   		If rst.Fields(8).Value <> 0 And rst.Fields(7).Value <> 0 Then ' Si el ciclo es no valido
   
   
   		VarC	= CInt(rst.Fields(6).Value) / 10
   		VarPR	= CInt(rst.Fields(7).Value)
   		
   		bfde4b54-0db7-4817-8032-87127bf19bb9 "VarC# " & VarC & " y VarPR " & VarPR
   			
   		
   			' Suma de formulas utilizadas
   			If LavadoraNro <> 4 Then
   				programaBraun(VarPR) = programaBraun(VarPR) + 1
   		If Err.Number <> 0 Then
   			bfde4b54-0db7-4817-8032-87127bf19bb9 "Error en S500 - en la asignacion de variables programaBraun en loop#" & Err.Number & " " & Err.Description
   			Err.Clear
   			Set conn = Nothing  
   			Exit Sub
   		End If
   				tCargaBraun(VarPR) = tCargaBraun(VarPR) + VarC
   		If Err.Number <> 0 Then
   			bfde4b54-0db7-4817-8032-87127bf19bb9 "Error en S500 - en la asignacion de variables tCargaBraun en loop#" & Err.Number & " " & Err.Description
   			Err.Clear
   			Set conn = Nothing  
   			Exit Sub
   		End If
   			Else
   				programaGirbau(VarPR) = programaGirbau(VarPR) + 1
   		If Err.Number <> 0 Then
   			bfde4b54-0db7-4817-8032-87127bf19bb9 "Error en S500 - en la asignacion de variables programaGirbau en loop#" & Err.Number & " " & Err.Description
   			Err.Clear
   			Set conn = Nothing  
   			Exit Sub
   		End If
   				tCargaGirbau(VarPR) = tCargaGirbau(VarPR) + VarC
   		If Err.Number <> 0 Then
   			bfde4b54-0db7-4817-8032-87127bf19bb9 "Error en S500 - en la asignacion de variables tCargaGirbau en loop#" & Err.Number & " " & Err.Description
   			Err.Clear
   			Set conn = Nothing  
   			Exit Sub
   		End If
   			End If
   			
   		End If
   		
   		rst.MoveNext
   		
   		If Err.Number <> 0 Then
   			bfde4b54-0db7-4817-8032-87127bf19bb9 "Error en S500 - en la asignacion de variables locales en loop#" & Err.Number & " " & Err.Description
   			Err.Clear
   			Set conn = Nothing  
   			Exit Sub
   		End If
   	Loop
   	
   	bfde4b54-0db7-4817-8032-87127bf19bb9 "Sale del loop de Lectura de registros S500 - de Lav nro " & LavadoraNro
   	
   	conn.close
   	Set rst = Nothing
   	Set conn = Nothing
   	
   Next
   
   bfde4b54-0db7-4817-8032-87127bf19bb9 "Sale del loop general de rst"
   
   '' %%%%%%%%%%%%%%%%%%%%%%%%%%%%%%%%%%%%%%%%%%%%%%%%%%%%%%%%%%%%%%%%%%%%%%%%%%%%%%%%%%%%%%%%%%%%%%%%%%%%%%%%%%%
   '' %%%%%%%%%%%%    IMPRESION DE DATOS EN INFORME    %%%%%%%%%%%%%%%%%%%%%%%%  XD  %%%%%%%%%%%%%%%%%%%%%%%%%%%%
   '' %%%%%%%%%%%%%%%%%%%%%%%%%%%%%%%%%%%%%%%%%%%%%%%%%%%%%%%%%%%%%%%%%%%%%%%%%%%%%%%%%%%%%%%%%%%%%%%%%%%%%%%%%%%
   
   Dim NameInfDiario
   
   
   If Err.Number <> 0 Then
   	bfde4b54-0db7-4817-8032-87127bf19bb9 "Cambio de nombre Informe Diario Lavs S500 - 2 Error #" & Err.Number & " " & Err.Description
   	Err.Clear 
   	Exit Sub
   End If
   
   ' Creacion devariables locales
   Dim objExcel
   Dim colMaquinadosBraun, colCantidadesBraun, colMaquinadosGirbau, colCantidadesGirbau
   Dim objfso
   
   'Asignacion inicial de variables locales
   colMaquinadosBraun	= 3
   colMaquinadosGirbau = 9
   colCantidadesBraun	= 4
   colCantidadesGirbau	= 10
   	
   'Creacion de Archivo .xls
   Set objExcel = CreateObject("Excel.Application")
   
   objExcel.Visible = False
   
   objExcel.Workbooks.Open "C:\ESPACIO DE TRABAJO\InformeDiario\Plantillas\InformeDiarioLavsMensual.xls"
   
   'Fin creacion archivo .xls
   If Err.Number <> 0 Then
   	bfde4b54-0db7-4817-8032-87127bf19bb9 "Error en  creacion de archivo: " & Err.Number & " :" & Err.Description
   	Err.Clear
   End If
   
   ' Imprimo tipo de informe
   objExcel.Cells(2,5).Value = impTipo
   
   objExcel.Cells(3,5).Value = impDesde
   objExcel.Cells(3,8).Value = impHasta
   						
   ' Inserción de datos en el informe
   
   'Datos de cantidad de programas
   For i = 0 To 14
   	
   	If i <= 9 Then
   		objExcel.Cells(i+7,colMaquinadosBraun).Value 	= programaBraun		(i + 1)
   		objExcel.Cells(i+7,colCantidadesBraun).Value 	= tCargaBraun		(i + 1)
   		objExcel.Cells(i+7,colMaquinadosGirbau).Value 	= programaGirbau	(i + 1)
   		objExcel.Cells(i+7,colCantidadesGirbau).Value 	= tCargaGirbau		(i + 1)
   	End If
   	
   If Err.Number <> 0 Then
   	bfde4b54-0db7-4817-8032-87127bf19bb9 "Error en Impresion de formulas 1ra en: " & i & " #" & Err.Number & " " & Err.Description
   	Err.Clear
   End If
   	
   	If i > 9 And i <= 11 Then
   		objExcel.Cells(i+12,colMaquinadosBraun).Value	= programaBraun		(i + 1)
   		objExcel.Cells(i+12,colCantidadesBraun).Value	= tCargaBraun		(i + 1)
   		objExcel.Cells(i+12,colMaquinadosGirbau).Value	= programaGirbau	(i + 1)
   		objExcel.Cells(i+12,colCantidadesGirbau).Value	= tCargaGirbau		(i + 1)
   	End If
   	
   If Err.Number <> 0 Then
   	bfde4b54-0db7-4817-8032-87127bf19bb9 "Error en Impresion de formulas 2da en: " & i & " #" & Err.Number & " " & Err.Description
   	Err.Clear
   End If
   	
   	If i > 11 Then
   		objExcel.Cells(i+5,colMaquinadosBraun).Value 	= programaBraun		(i + 1)
   		objExcel.Cells(i+5,colCantidadesBraun).Value 	= tCargaBraun		(i + 1)
   		objExcel.Cells(i+5,colMaquinadosGirbau).Value 	= programaGirbau	(i + 1)
   		objExcel.Cells(i+5,colCantidadesGirbau).Value 	= tCargaGirbau		(i + 1)
   		
   	End If
   	
   If Err.Number <> 0 Then
   	bfde4b54-0db7-4817-8032-87127bf19bb9 "Error en Impresion de formulas 3ra en: " & i & " #" & Err.Number & " " & Err.Description
   	Err.Clear
   End If
   Next
   
   If Err.Number <> 0 Then
   	bfde4b54-0db7-4817-8032-87127bf19bb9 "Error en Impresion de formulas#" & Err.Number & " " & Err.Description
   	Err.Clear
   End If
   
   ' Fin de impresion de datos en tabla
   Dim Text
   Select Case tipo_Inf
   	Case 0 ' Periodico
   		Text = "Informe_Periodico"
   	Case 1
   		Text = "Informe_Mensual"
   	Case 2
   		Text = "Informe_Anual"	
   End Select
   
   NameInfDiario = "C:\ESPACIO DE TRABAJO\InformeDiario\" & Text & "_Lavs" &(Replace(CStr(Date),"/","")&Replace(CStr(Time),":",""))&".xls"
   
   objExcel.ActiveWorkbook.SaveAs NameInfDiario, 56
   objExcel.ActiveWorkbook.Close
   objExcel.Application.Quit
   
   
   Set objfso = CreateObject("Scripting.FileSystemObject")
   Do While objfso.FileExists(NameInfDiario) = False
   Loop
   k = Timer +5
   Do While (Timer<k)
   Loop	
   
   	If Err.Number <> 0 Then
   		bfde4b54-0db7-4817-8032-87127bf19bb9 "Error en creacion de archivo excel#" & Err.Number & " " & Err.Description
   		Err.Clear
   	End If
   
   bfde4b54-0db7-4817-8032-87127bf19bb9 "NameInfDiario#" & CStr(NameInfDiario)
   
   '## ENVIAR INFORME POR EMAIL
   
   Dim appOutlook 'As OUTLOOK.APPLICATION
   Dim mlNewMail 'As MailItem
   Dim objEntry
   
   
   Const addressee = "crj@eprocsrl.com.ar; danielst@live.com.ar; josemariacullen@hotmail.com;"' zekeserio@hotmail.com;"
   
   Set appOutlook = CreateObject("OUTLOOK.APPLICATION")
   
   
   'Generating and sending an e-mail:
   Set mlNewMail = appOutlook.CreateItem(0)
   mlNewMail.Display
   mlNewMail.To = addressee
   mlNewMail.Subject = Text + " de produccion"
   mlNewMail.Body = Text
   
   mlNewMail.Attachments.Add CStr(NameInfDiario)
   
   mlNewMail.save
   mlNewMail.send 
   
   'Error routine
   If Err.Number <> 0 Then
   	bfde4b54-0db7-4817-8032-87127bf19bb9 "Error al enviar el email #" & Err.Number & " " & Err.Description
   End If

VB script "S404_ActMes"
   	Dim mesAnterior
   
   	mesAnterior = Date()
   
   	mesAnterior = DateAdd("m",-1, mesAnterior)
   	
   	SmartTags("Inf_Mes") = Month(mesAnterior)
   	

VB script "S405_ActAno"
   	Dim anoAnterior
   
   	anoAnterior = Date()
   
   	anoAnterior = DateAdd("yyyy",-1, anoAnterior)
   	
   	SmartTags("Inf_Ano") = Year(anoAnterior)
   	

VB script "S406_UltimoDiaDelMes"
   Dim bisiesto
   
   ' verificar que el año sea bisiesto
   If (ano Mod 4) = 0 And ((ano Mod 100) <> 0 Or (ano Mod 400) = 0) Then
   	bisiesto = 1
   Else
   	bisiesto = 0
   End If
   
   If mes = 1 Or mes = 3 Or mes = 5 Or mes = 7 Or mes = 8 Or mes = 10 Or mes = 12 Then
   	S406_UltimoDiaDelMes = 31
   End If
   
   If mes = 4 Or mes = 6 Or mes = 9 Or mes = 11 Then
   	S406_UltimoDiaDelMes = 30
   End If
   
   If bisiesto = 1 And mes = 2 Then
   	S406_UltimoDiaDelMes = 29
   End If
   
   If bisiesto = 0 And mes = 2 Then
   	S406_UltimoDiaDelMes = 28
   End If

VB script "I100_LeerIndice"
   'Declaracion de Variables locales
   Dim conn, rst, SQL_Table
   
   On Error Resume Next
   
   Set conn = CreateObject("ADODB.Connection")
   Set rst = CreateObject("ADODB.Recordset")
   
   'Abrir BDD
   conn.Open "Provider=MSDASQL;Initial Catalog=Lavadero;DSN=Lavadero"
   
   
   'Chequeo de error
   If Err.Number <> 0 Then
   	bfde4b54-0db7-4817-8032-87127bf19bb9 "Error #" & Err.Number & " " & Err.Description
   	Err.Clear 
   	Set conn = Nothing
   	Exit Sub
   End If
   
   
   SQL_Table = "SELECT * FROM indicesPlanchas WHERE  ID = '" & SmartTags("Idx_ID") &"';"
   
   'Ejecutar consulta
   Set rst = conn.Execute(SQL_Table)
   
   SmartTags("Idx_Name") = rst.Fields(1).Value
   
   rst.close 
   
   conn.close
   
   Set rst = Nothing
   Set conn = Nothing

VB script "I101_EscribirIndice"
   'Declaracion de variables locales
   Dim conn, rst, SQL_Table, fechapl, fecha, hora
   
   On Error Resume Next
   
   Set conn = CreateObject("ADODB.Connection")
   Set rst = CreateObject("ADODB.Recordset")
   
   'Abrir BBDD
   conn.Open "Provider=MSDASQL;Initial Catalog=Lavadero;DSN=Lavadero"
   'conn.Open "Provider=MSDASQL;Initial Catalog=" & SmartTags("szDatabase") & ";DSN="&Database_Name&"" 'DSN= name of the odbc database - DSN= Name der ODBC-Datenbank
   
   
   
   'Crear consulta de insersion
   SQL_Table = "INSERT INTO indicesPlanchas VALUES ('"_
   		& SmartTags("Idx_ID_Nuevo")_
   		& "' , '" & SmartTags("Idx_Name_Nuevo") & "')"
   
   Set rst = conn.Execute(SQL_Table)
   
   'Error routine - Fehlerroutine
   If Err.Number <> 0 Then
   	bfde4b54-0db7-4817-8032-87127bf19bb9 "Error abrirb base #" & Err.Number & " " & Err.Description
   	Err.Clear
   	Set conn = Nothing 
   	Exit Sub
   End If
   
   conn.close
   
   Set rst = Nothing
   Set conn = Nothing

VB script "I102_CambiarIndice"
   'Declaracion de variables locales
   Dim conn, rst, SQL_Table
   
   On Error Resume Next
   
   Set conn = CreateObject("ADODB.Connection")
   Set rst = CreateObject("ADODB.Recordset")
   
   'Abrir BBDD
   conn.Open "Provider=MSDASQL;Initial Catalog=Lavadero;DSN=Lavadero"
   
   'Crear consulta de insersion
   SQL_Table = "UPDATE indicesPlanchas SET indice = '"_
   		& SmartTags("Idx_Name_Cambiar")_
   		& "' WHERE Cant = '" & SmartTags("Idx_ID_Cambiar") & "';"
   
   Set rst = conn.Execute(SQL_Table)
   
   'Error routine - Fehlerroutine
   If Err.Number <> 0 Then
   	bfde4b54-0db7-4817-8032-87127bf19bb9 "Error abrirb base #" & Err.Number & " " & Err.Description
   	Err.Clear
   	Set conn = Nothing 
   	Exit Sub
   End If
   
   conn.close
   
   Set rst = Nothing
   Set conn = Nothing

VB script "I103_ActualizarIndice"
   'Declaracion de Variables locales
   Dim conn, rst, SQL_Table
   
   On Error Resume Next
   
   Set conn = CreateObject("ADODB.Connection")
   Set rst = CreateObject("ADODB.Recordset")
   
   'Abrir BDD
   conn.Open "Provider=MSDASQL;Initial Catalog=Lavadero;DSN=Lavadero"
   
   
   'Chequeo de error
   If Err.Number <> 0 Then
   	bfde4b54-0db7-4817-8032-87127bf19bb9 "Error #" & Err.Number & " " & Err.Description
   	Err.Clear 
   	Set conn = Nothing
   	Exit Sub
   End If
   
   If (SmartTags("Idx_ID_1") <= 0) Then
   	SmartTags("Idx_ID_1") = 1
   End If
   
   SQL_Table = "SELECT * FROM indicesPlanchas WHERE Cant >= '" & SmartTags("Idx_ID_1") &"' ORDER BY Cant;"
   
   'Ejecutar consulta
   Set rst = conn.Execute(SQL_Table)
   
   
   'Llenado de variables que muestan la lista
   If rst.EOF = False Then
   	SmartTags("Idx_ID_1") = rst.Fields(0).Value
   	SmartTags("Idx_Name_1") = rst.Fields(1).Value
   	rst.MoveNext
   Else
   	SmartTags("Idx_ID_1") = 0
   	SmartTags("Idx_Name_1") = "Vacio"
   End If
   
   If rst.EOF = False Then
   	SmartTags("Idx_ID_2") = rst.Fields(0).Value
   	SmartTags("Idx_Name_2") = rst.Fields(1).Value
   	rst.MoveNext
   Else
   	SmartTags("Idx_ID_2") = 0
   	SmartTags("Idx_Name_2") = "Vacio"
   End If
   
   If rst.EOF = False Then
   	SmartTags("Idx_ID_3") = rst.Fields(0).Value
   	SmartTags("Idx_Name_3") = rst.Fields(1).Value
   	rst.MoveNext
   Else
   	SmartTags("Idx_ID_3") = 0
   	SmartTags("Idx_Name_3") = "Vacio"
   End If
   
   If rst.EOF = False Then
   	SmartTags("Idx_ID_4") = rst.Fields(0).Value
   	SmartTags("Idx_Name_4") = rst.Fields(1).Value
   	rst.MoveNext
   Else
   	SmartTags("Idx_ID_4") = 0
   	SmartTags("Idx_Name_4") = "Vacio"
   End If
   
   If rst.EOF = False Then
   	SmartTags("Idx_ID_5") = rst.Fields(0).Value
   	SmartTags("Idx_Name_5") = rst.Fields(1).Value
   	rst.MoveNext
   Else
   	SmartTags("Idx_ID_5") = 0
   	SmartTags("Idx_Name_5") = "Vacio"
   End If
   
   
   rst.close
   
   conn.close
   
   Set rst = Nothing
   Set conn = Nothing

VB script "S501_InformePer_Planchas"
   'Declaration of local tags - Deklaration von lokalem Variablen
   Dim conn, rst, SQL_Table, i, j
   
   Dim Consulta,where, mesdesde, meshasta, diadesde, diahasta
   Dim impDesde, impHasta, impTipo
   
   On Error Resume Next
   
   Set conn = CreateObject("ADODB.Connection")
   Set rst = CreateObject("ADODB.Recordset")
   
   'Open data source - Datenquelle öffnen
   conn.Open "Provider=MSDASQL;Initial Catalog=Lavadero;DSN=Lavadero"
   'Error routine - Fehlerroutine
   If Err.Number <> 0 Then
   	bfde4b54-0db7-4817-8032-87127bf19bb9 "Conexion Error #" & Err.Number & " " & Err.Description
   	Err.Clear
   	conn.close
   	Set conn = Nothing
   	Exit Sub
   End If
   
   '///////// ARMADO DE WCLAUSULA   ///////////////
   Select Case tipo_Inf
   	Case 0 ' Periodico
   		
   		If Month(desde) < 10 Then
   			mesdesde = "0" + CStr(Month(desde))
   		Else
   			mesdesde = CStr(Month(desde))
   		End If
   		
   		If Month(hasta) < 10 Then
   			meshasta = "0" + CStr(Month(hasta))
   		Else
   			meshasta = CStr(Month(hasta))
   		End If
   		
   		If Day(desde) < 10 Then
   			diadesde = "0" + CStr(Day(desde))
   		Else
   			diadesde = CStr(Day(desde))
   		End If
   		
   		If Day(hasta) < 10 Then
   			diahasta = "0" + CStr(Day(hasta))
   		Else
   			diahasta = CStr(Day(hasta))
   		End If
   			
   		where =" WHERE cast(fecha As Date) >= '"
   		where = where & CStr(Year(desde)) & "-" & mesdesde & "-" & diadesde & "' "
   		where = where & "and cast(fecha As Date) <= '"
   		where = where & CStr(Year(hasta)) & "-" & meshasta & "-" & diahasta & "' "
   		where = where & " order by fecha"
   		
   		impDesde = CStr(Year(desde)) & "-" & mesdesde & "-" & diadesde
   		impHasta = CStr(Year(hasta)) & "-" & meshasta & "-" & diahasta
   		impTipo = "Periodico"
   		
   	Case 1 'Mensual
   		If hasta < 10 Then
   			meshasta = "0" + CStr(hasta)
   		Else
   			meshasta = CStr(hasta)
   		End If
   		
   		where = " WHERE cast(fecha As Date) like '%"
   		where = where & CStr(desde) & "-" & meshasta & "%' "
   		where = where & "order by fecha"
   		
   		impDesde = CStr(desde) & "-" & meshasta & "-01"
   		impHasta = CStr(desde) & "-" & meshasta & "-" & CStr(S406_UltimoDiaDelMes(meshasta,desde))
   		impTipo = "Mensual"
   		
   	Case 2 'Anual
   		
   		where = " WHERE cast(fecha As Date) like '%"
   		where = where & CStr(hasta) & "-%' "
   		where = where & "order by fecha"
   		
   		impDesde = CStr(hasta) & "-01-01"
   		impHasta = CStr(hasta) & "-12-31"
   		impTipo = "Anual"
   		
   End Select
   
   If Err.Number <> 0 Then
   	bfde4b54-0db7-4817-8032-87127bf19bb9 "Consulta Lav Error 3#" & Err.Number & " " & Err.Description
   	Err.Clear
   	'Close data source
   	Set conn = Nothing
   	Set rst = Nothing 
   	Exit Sub
   End If
   
   
   ' #################   Generacion de consulta a BDD Plancha1   ######################
   
   Dim DiaAnterior
   DiaAnterior = Date()
   
   ' Datos para el informe
   SmartTags("Inf_FechaInforme") 			= DiaAnterior
   SmartTags("Inf_FechaInforme_WeekDay") 	= Weekday(DiaAnterior)
   
   Consulta = "SELECT * FROM resultadosDiariosPlanchadoras" & where
   
   'Execute
   Set rst = conn.Execute(Consulta)
   
   'Error routine
   If Err.Number <> 0 Then
   	bfde4b54-0db7-4817-8032-87127bf19bb9 "Consulta1 PL1 Error #" & Err.Number & " " & Err.Description
   	Err.Clear
   	'Close data source - Datenquelle schließen0
   	conn.close
   	Set conn = Nothing
   	Set rst = Nothing 
   	Exit Sub
   End If
   	
   '####################### PROCESAMIENTO DE DATOS PLANCHA 1 ########################
   
       Dim diasTotal(5),horasTotal(5)	, strTotal(5)
       Dim diasProd(5)	,horasProd(5)	, strProd(5)
       Dim diasRend(5)	,horasRend(5)	, strRend(5)
   
       Dim personasProm(5)
       Dim cantDias
       Dim indiceProm(5)
               
       Dim XProd(5)
       Dim XRend(5)
       Dim tmp_1
       
       Dim valorDecimal, parteEntera, parteDecimal
       
       For i = 1 To 5
   		personasProm	(i) = 0.0
   		horasTotal		(i)	= 0.0
   		horasProd		(i) = 0.0
   		horasRend		(i) = 0.0
   		indiceProm		(i) = 0.0
   		XProd			(i) = 0.0
      		XRend			(i) = 0.0
   	Next
   	
   	cantDias = 0
       
       
       'Entra a recorrer la consutla, el RST
       Do While rst.EOF = False
   		
   		j = 4
   		If CDbl(rst.Fields(j).Value) >= 0 Then
   			cantDias = cantDias + 1
   			
   	      
   	        For i = 2 To 5
   		        horasTotal(i)	= horasTotal(i)	 	+ CDbl(rst.Fields(j).Value)
   		        j = j + 1
   		        horasProd(i) 	= horasProd(i) 		+ CDbl(rst.Fields(j).Value)
   		        j = j + 1
   		        horasRend(i) 	= horasRend(i)		+ CDbl(rst.Fields(j).Value)
   		        j = j + 1
   		        personasProm(i) = personasProm(i) 	+ CDbl(rst.Fields(j).Value)
   		        j = j + 1
   			Next
   		
   		End If
   		
           rst.MoveNext
           
   	Loop  
   	
   	If Err.Number <> 0 Then
   		bfde4b54-0db7-4817-8032-87127bf19bb9 "Recoleccion de Datos2 Periodico Planchas Error #" & Err.Number & " " & Err.Description
   		Err.Clear
   		Exit Sub
   	End If       
       
       'Calculo de tiempos totales
       For i = 2 To 5
           horasTotal	(i) = horasTotal(i) * 24.0
           horasProd	(i) = horasProd(i)	* 24.0
           horasRend	(i) = horasRend(i) 	* 24.0
           
           If cantDias <> 0 Then
           	personasProm(i) = Int(personasProm(i)/ cantDias)
   		End If
   	Next
   	
       For i = 2 To 5
           horasTotal	(1) = horasTotal	(1) + horasTotal	(i)
           horasProd	(1) = horasProd		(1) + horasProd		(i)
           horasRend	(1) = horasRend		(1) + horasRend		(i) 
   		personasProm(1) = personasProm	(1) + personasProm	(i)
   	Next
   	
   	personasProm(1) = Int(personasProm(1))
   	
   	
       For i = 1 To 5
           'Obtengo los porcentajes de tiempos
           
          	If horasTotal(i) <> 0 Then
               XProd(i) = 100.0 * (horasProd(i) / horasTotal(i))
           Else    
               XProd(i) = 0.0
   		End If
   		
           If horasProd(i) <> 0 Then
               XRend(i) = 100.0 * (horasRend(i) / horasProd(i))
   		Else
   			XRend(i) = 0.0
   		End If
   	Next
           
   	If Err.Number <> 0 Then
   		bfde4b54-0db7-4817-8032-87127bf19bb9 "Procesamiento final Datos Informe PEriodico Plancha Error #" & Err.Number & " " & Err.Description
   		Err.Clear
   		Exit Sub
   	End If
   
   conn.close
   Set rst = Nothing
   Set conn = Nothing
   
   ' Pasaje de diashoras  a horas
   		
   For i= 1 To 5
   	diasTotal(i) 	= Fix(horasTotal(i)) / 1
   	horasTotal(i) 	= horasTotal(i) - diasTotal(i)
   	strTotal(i) 	= SA2_TotalTimeToString(diasTotal(i), horasTotal(i))
   	
   	
   	diasProd(i) 	= Fix(horasProd(i)) / 1
   	horasProd(i) 	= horasProd(i) - diasProd(i)
   	strProd(i) 		= SA2_TotalTimeToString(diasProd(i), horasProd(i))
   	
   	
   	diasRend(i) 	= Fix(horasRend(i)) / 1
   	horasRend(i)	= horasRend(i) - diasRend(i)
   	strRend(i) 		= SA2_TotalTimeToString(diasRend(i), horasRend(i))
   Next
   
   
   '///////////////////////////////     Extraccion de Indices   /////////////////
   Dim connindx, rstindx, Consultaindx, listaIndices(60), k, indice(5)
   
   Set connindx = CreateObject("ADODB.Connection")
   Set rstindx = CreateObject("ADODB.Recordset")
   
   'Open data source - Datenquelle öffnen
   connindx.Open "Provider=MSDASQL;Initial Catalog=Lavadero;DSN=Lavadero"
   'Error routine - Fehlerroutine
   If Err.Number <> 0 Then
   	bfde4b54-0db7-4817-8032-87127bf19bb9 "Conexion Error a indicesPlanchas" & Err.Number & " " & Err.Description
   	Err.Clear
   	Set connindx = Nothing  
   	Exit Sub
   End If
   
   Consultaindx = "SELECT * FROM indicesPlanchas;"
   
   'Ejecutar consulta
   Set rstindx = connindx.Execute(Consultaindx)
   
   ' Establecer los indices
   j = 1
   k = 1
   Do While rstindx.EOF = False
   	For j = 1 To 5
   		If (rstindx.Fields(0).Value = personasProm(j)) Then ' Si el ciclo es no valido
   			indice(j) = rstindx.Fields(1).Value / 10.0
   		End If
   	Next
   	
   	'Para imprimir todos los indices
   	listaIndices(k) = rstindx.Fields(1).Value / 10.0
   	k = k + 1
   	
   	rstindx.MoveNext
   Loop
   
   If Err.Number <> 0 Then
   	bfde4b54-0db7-4817-8032-87127bf19bb9 "Error en establecer los operadores InfPreiodico Planchas#" & Err.Number & " " & Err.Description
   	Err.Clear
   	Set connindx = Nothing  
   	Exit Sub
   End If
   
   'Creo Excel
   Dim objExcel, fila
   
   fila = 5
   Set objExcel = CreateObject("Excel.Application")
   
   objExcel.Visible = False
   
   objExcel.Workbooks.Open "C:\ESPACIO DE TRABAJO\InformeDiario\Plantillas\InformeDiarioExcelP.xlsx"
       
       ' Fecha informe
   	objExcel.Cells(2,4).Value 		= DiaAnterior
   
       'Grales
       objExcel.Cells(fila,2).Value 		= strTotal		(1)
       objExcel.Cells(fila,3).Value 		= strProd 		(1)
       objExcel.Cells(fila,4).Value 		= XProd			(1)
   	objExcel.Cells(fila,5).Value 		= strRend		(1)
   	objExcel.Cells(fila,6).Value 		= XRend			(1)
   	objExcel.Cells(fila,7).Value 		= personasProm	(1)
   	objExcel.Cells(fila,8).Value 		= indice 		(1)
   	
   If Err.Number <> 0 Then
   	bfde4b54-0db7-4817-8032-87127bf19bb9 "Asignasion Datos Informe Plancha Periodico Error #" & Err.Number & " " & Err.Description
   	Err.Clear 
   End If
   
   	'Supervisores
   For i = 1 To 4 
   	
   	objExcel.Cells(i+fila,2).Value 		= strTotal		(i+1)
   	objExcel.Cells(i+fila,3).Value 		= strProd		(i+1)
   	objExcel.Cells(i+fila,4).Value 		= XProd			(i+1)
   	objExcel.Cells(i+fila,5).Value 		= strRend		(i+1)
   	objExcel.Cells(i+fila,6).Value	    = XRend			(i+1)
   	objExcel.Cells(i+fila,7).Value	    = personasProm	(i+1)
   	objExcel.Cells(i+fila,8).Value 		= indice 		(i+1)
   	
   	
   	If Err.Number <> 0 Then
   		bfde4b54-0db7-4817-8032-87127bf19bb9 "Asignasion Datos Sup"& CStr(i) &" PL1 Error #" & Err.Number & " " & Err.Description
   		Err.Clear 
   	End If
   Next
   
   For j = 1 To 4
   	If 0 = personasProm(j+1) Then
   		objExcel.Cells(j+fila,9).Value = 1
   	End If
   Next
   
   'Lista de indices
   For i = 1 To 15 
   	objExcel.Cells(i+4,13).Value 	= listaIndices (i)
   	objExcel.Cells(i+4,15).Value 	= listaIndices (i+15)
   Next
   
   Dim NameInfDiario, Text
   
   ' Text to be sent 
   Select Case tipo_Inf
   	Case 0 ' Periodico
   		Text = "Informe Periodico"
   	Case 1
   		Text = "Informe Mensual"
   	Case 2
   		Text = "Informe Anual"	
   End Select
   
   NameInfDiario = "C:\ESPACIO DE TRABAJO\InformeDiario\" & Text & "_Pla"&(Replace(CStr(Date),"/","")&Replace(CStr(Time),":",""))&".xlsx"
   
   objExcel.ActiveWorkbook.SaveAs NameInfDiario
   objExcel.ActiveWorkbook.Close
   objExcel.Application.Quit
   	
   '#########################################################
   
   
   '## ENVIAR INFORME POR EMAIL
   
   Dim appOutlook 'As OUTLOOK.APPLICATION
   Dim mlNewMail 'As MailItem
   Dim objEntry
   
   Const addressee = "crj@eprocsrl.com.ar; danielst@live.com.ar; josemariacullen@hotmail.com;"' zekeserio@hotmail.com;"
   
   
   Set appOutlook = CreateObject("OUTLOOK.APPLICATION")
   
   'Generating and sending an e-mail:
   Set mlNewMail = appOutlook.CreateItem(0)
   mlNewMail.Display
   mlNewMail.To = addressee
   mlNewMail.Subject = Text + " de produccion"
   mlNewMail.Body = Text
   
   mlNewMail.Attachments.Add CStr(NameInfDiario)
   
   mlNewMail.save
   mlNewMail.send 
   
   'Error routine
   If Err.Number <> 0 Then
   	bfde4b54-0db7-4817-8032-87127bf19bb9 "Error al enviar el email Inf periodico #" & Err.Number & " " & Err.Description
   End If

VB script "S407_Act_IndicePLC"
   'Declaracion de Variables locales
   Dim conn, rst, SQL_Table
   
   On Error Resume Next
   
   Set conn = CreateObject("ADODB.Connection")
   Set rst = CreateObject("ADODB.Recordset")
   
   'Abrir BDD
   conn.Open "Provider=MSDASQL;Initial Catalog=Lavadero;DSN=Lavadero"
   
   
   'Chequeo de error
   If Err.Number <> 0 Then
   	bfde4b54-0db7-4817-8032-87127bf19bb9 "Error #" & Err.Number & " " & Err.Description
   	Err.Clear 
   	Set conn = Nothing
   	Exit Sub
   End If
   
   
   SQL_Table = "SELECT * FROM indicesPlanchas WHERE  Cant = '" & SmartTags("Planchadora1_SumaOperario") &"';"
   
   'Ejecutar consulta
   Set rst = conn.Execute(SQL_Table)
   
   SmartTags("Indices_objetivo_100") = CDbl(rst.Fields(1).Value) / 10
   
   rst.close
   
   conn.close
   
   Set rst = Nothing
   Set conn = Nothing

VB script "S600_Cambiar_Vars_Todos"
   Dim progStr
   
   Select Case Lav
   	Case 1
   		progStr = CStr(SmartTags("_Prog_aModifBraun"))
   		Select Case Parametro
   			Case 1
   				SmartTags("Lav1_Prog"&progStr&"_EnjIni_Cant") = SmartTags("_Prog_EnjIni_Cant")
   				SmartTags("Lav2_Prog"&progStr&"_EnjIni_Cant") = SmartTags("_Prog_EnjIni_Cant")
   				SmartTags("Lav3_Prog"&progStr&"_EnjIni_Cant") = SmartTags("_Prog_EnjIni_Cant")
   			Case 2
   				SmartTags("Lav1_Prog"&progStr&"_EnjIni_Tiempo") = SmartTags("_Prog_EnjIni_Tiempo")
   				SmartTags("Lav2_Prog"&progStr&"_EnjIni_Tiempo") = SmartTags("_Prog_EnjIni_Tiempo")
   				SmartTags("Lav3_Prog"&progStr&"_EnjIni_Tiempo") = SmartTags("_Prog_EnjIni_Tiempo")
   			Case 3
   				SmartTags("Lav1_Prog"&progStr&"_EnjIni_NivAg") = SmartTags("_Prog_EnjIni_NivAg")
   				SmartTags("Lav2_Prog"&progStr&"_EnjIni_NivAg") = SmartTags("_Prog_EnjIni_NivAg")
   				SmartTags("Lav3_Prog"&progStr&"_EnjIni_NivAg") = SmartTags("_Prog_EnjIni_NivAg")
   			Case 4
   				SmartTags("Lav1_Prog"&progStr&"_PreLav_Tiempo") = SmartTags("_Prog_PreLav_Tiempo")
   				SmartTags("Lav2_Prog"&progStr&"_PreLav_Tiempo") = SmartTags("_Prog_PreLav_Tiempo")
   				SmartTags("Lav3_Prog"&progStr&"_PreLav_Tiempo") = SmartTags("_Prog_PreLav_Tiempo")
   			Case 5
   				SmartTags("Lav1_Prog"&progStr&"_PreLav_NivAg") = SmartTags("_Prog_PreLav_NivAg")
   				SmartTags("Lav2_Prog"&progStr&"_PreLav_NivAg") = SmartTags("_Prog_PreLav_NivAg")
   				SmartTags("Lav3_Prog"&progStr&"_PreLav_NivAg") = SmartTags("_Prog_PreLav_NivAg")
   			Case 6
   				SmartTags("Lav1_Prog"&progStr&"_PreLav_AgCaliente") = SmartTags("_Prog_PreLav_AgCaliente")
   				SmartTags("Lav2_Prog"&progStr&"_PreLav_AgCaliente") = SmartTags("_Prog_PreLav_AgCaliente")
   				SmartTags("Lav3_Prog"&progStr&"_PreLav_AgCaliente") = SmartTags("_Prog_PreLav_AgCaliente")
   			Case 7
   				SmartTags("Lav1_Prog"&progStr&"_PreLav_Vapor") = SmartTags("_Prog_PreLav_Vapor")
   				SmartTags("Lav2_Prog"&progStr&"_PreLav_Vapor") = SmartTags("_Prog_PreLav_Vapor")
   				SmartTags("Lav3_Prog"&progStr&"_PreLav_Vapor") = SmartTags("_Prog_PreLav_Vapor")
   			Case 8
   				SmartTags("Lav1_Prog"&progStr&"_PreLav_Temperatura") = SmartTags("_Prog_PreLav_Temperatura")
   				SmartTags("Lav2_Prog"&progStr&"_PreLav_Temperatura") = SmartTags("_Prog_PreLav_Temperatura")
   				SmartTags("Lav3_Prog"&progStr&"_PreLav_Temperatura") = SmartTags("_Prog_PreLav_Temperatura")
   			Case 9
   				SmartTags("Lav1_Prog"&progStr&"_Lav1_Tiempo") = SmartTags("_Prog_Lav1_Tiempo")
   				SmartTags("Lav2_Prog"&progStr&"_Lav1_Tiempo") = SmartTags("_Prog_Lav1_Tiempo")
   				SmartTags("Lav3_Prog"&progStr&"_Lav1_Tiempo") = SmartTags("_Prog_Lav1_Tiempo")
   			Case 10
   				SmartTags("Lav1_Prog"&progStr&"_Lav1_NivAg") = SmartTags("_Prog_Lav1_NivAg")
   				SmartTags("Lav2_Prog"&progStr&"_Lav1_NivAg") = SmartTags("_Prog_Lav1_NivAg")
   				SmartTags("Lav3_Prog"&progStr&"_Lav1_NivAg") = SmartTags("_Prog_Lav1_NivAg")
   			Case 11
   				SmartTags("Lav1_Prog"&progStr&"_Lav1_AgCaliente") = SmartTags("_Prog_Lav1_AgCaliente")
   				SmartTags("Lav2_Prog"&progStr&"_Lav1_AgCaliente") = SmartTags("_Prog_Lav1_AgCaliente")
   				SmartTags("Lav3_Prog"&progStr&"_Lav1_AgCaliente") = SmartTags("_Prog_Lav1_AgCaliente")
   			Case 12
   				SmartTags("Lav1_Prog"&progStr&"_Lav1_Temperatura") = SmartTags("_Prog_Lav1_Temperatura")
   				SmartTags("Lav2_Prog"&progStr&"_Lav1_Temperatura") = SmartTags("_Prog_Lav1_Temperatura")
   				SmartTags("Lav3_Prog"&progStr&"_Lav1_Temperatura") = SmartTags("_Prog_Lav1_Temperatura")
   			Case 13
   				SmartTags("Lav1_Prog"&progStr&"_Lav2_Tiempo") = SmartTags("_Prog_Lav2_Tiempo")
   				SmartTags("Lav2_Prog"&progStr&"_Lav2_Tiempo") = SmartTags("_Prog_Lav2_Tiempo")
   				SmartTags("Lav3_Prog"&progStr&"_Lav2_Tiempo") = SmartTags("_Prog_Lav2_Tiempo")
   			Case 14
   				SmartTags("Lav1_Prog"&progStr&"_Lav2_NivAg") = SmartTags("_Prog_Lav2_NivAg")
   				SmartTags("Lav2_Prog"&progStr&"_Lav2_NivAg") = SmartTags("_Prog_Lav2_NivAg")
   				SmartTags("Lav3_Prog"&progStr&"_Lav2_NivAg") = SmartTags("_Prog_Lav2_NivAg")
   			Case 15
   				SmartTags("Lav1_Prog"&progStr&"_Lav2_AgCaliente") = SmartTags("_Prog_Lav2_AgCaliente")	
   				SmartTags("Lav2_Prog"&progStr&"_Lav2_AgCaliente") = SmartTags("_Prog_Lav2_AgCaliente")	
   				SmartTags("Lav3_Prog"&progStr&"_Lav2_AgCaliente") = SmartTags("_Prog_Lav2_AgCaliente")		
   			Case 16
   				SmartTags("Lav1_Prog"&progStr&"_Lav2_Temperatura") = SmartTags("_Prog_Lav2_Temperatura")
   				SmartTags("Lav2_Prog"&progStr&"_Lav2_Temperatura") = SmartTags("_Prog_Lav2_Temperatura")
   				SmartTags("Lav3_Prog"&progStr&"_Lav2_Temperatura") = SmartTags("_Prog_Lav2_Temperatura")
   			Case 17
   				SmartTags("Lav1_Prog"&progStr&"_EnjFin_Cant") = SmartTags("_Prog_EnjFin_Cant")
   				SmartTags("Lav2_Prog"&progStr&"_EnjFin_Cant") = SmartTags("_Prog_EnjFin_Cant")
   				SmartTags("Lav3_Prog"&progStr&"_EnjFin_Cant") = SmartTags("_Prog_EnjFin_Cant")
   			Case 18
   				SmartTags("Lav1_Prog"&progStr&"_EnjFin_Tiempo") = SmartTags("_Prog_EnjFin_Tiempo")
   				SmartTags("Lav2_Prog"&progStr&"_EnjFin_Tiempo") = SmartTags("_Prog_EnjFin_Tiempo")
   				SmartTags("Lav3_Prog"&progStr&"_EnjFin_Tiempo") = SmartTags("_Prog_EnjFin_Tiempo")
   			Case 19
   				SmartTags("Lav1_Prog"&progStr&"_Centr_Tiempo") = SmartTags("_Prog_Centr_Tiempo")
   				SmartTags("Lav2_Prog"&progStr&"_Centr_Tiempo") = SmartTags("_Prog_Centr_Tiempo")
   				SmartTags("Lav3_Prog"&progStr&"_Centr_Tiempo") = SmartTags("_Prog_Centr_Tiempo")
   							
   		End Select 
   		
   		
   	Case 2
   		progStr = CStr(SmartTags("_Prog_aModifGirbau"))
   		Select Case Parametro
   			Case 1
   				SmartTags("Lav4_Prog"&progStr&"_EnjIni_Cant") = SmartTags("_Prog_EnjIni_Cant")
   			Case 2
   				SmartTags("Lav4_Prog"&progStr&"_EnjIni_Tiempo") = SmartTags("_Prog_EnjIni_Tiempo")
   			Case 3
   				SmartTags("Lav4_Prog"&progStr&"_EnjIni_NivAg") = SmartTags("_Prog_EnjIni_NivAg")
   			Case 4
   				SmartTags("Lav4_Prog"&progStr&"_PreLav_Tiempo") = SmartTags("_Prog_PreLav_Tiempo")
   			Case 5
   				SmartTags("Lav4_Prog"&progStr&"_PreLav_NivAg") = SmartTags("_Prog_PreLav_NivAg")
   			Case 6
   				SmartTags("Lav4_Prog"&progStr&"_PreLav_AgCaliente") = SmartTags("_Prog_PreLav_AgCaliente")
   			Case 7
   				SmartTags("Lav4_Prog"&progStr&"_PreLav_Vapor") = SmartTags("_Prog_PreLav_Vapor")
   			Case 8
   				SmartTags("Lav4_Prog"&progStr&"_PreLav_Temperatura") = SmartTags("_Prog_PreLav_Temperatura")
   			Case 9
   				SmartTags("Lav4_Prog"&progStr&"_Lav1_Tiempo") = SmartTags("_Prog_Lav1_Tiempo")
   			Case 10
   				SmartTags("Lav4_Prog"&progStr&"_Lav1_NivAg") = SmartTags("_Prog_Lav1_NivAg")
   			Case 11
   				SmartTags("Lav4_Prog"&progStr&"_Lav1_AgCaliente") = SmartTags("_Prog_Lav1_AgCaliente")
   			Case 12
   				SmartTags("Lav4_Prog"&progStr&"_Lav1_Temperatura") = SmartTags("_Prog_Lav1_Temperatura")
   			Case 13
   				SmartTags("Lav4_Prog"&progStr&"_Lav2_Tiempo") = SmartTags("_Prog_Lav2_Tiempo")
   			Case 14
   				SmartTags("Lav4_Prog"&progStr&"_Lav2_NivAg") = SmartTags("_Prog_Lav2_NivAg")
   			Case 15
   				SmartTags("Lav4_Prog"&progStr&"_Lav2_AgCaliente") = SmartTags("_Prog_Lav2_AgCaliente")		
   			Case 16
   				SmartTags("Lav4_Prog"&progStr&"_Lav2_Temperatura") = SmartTags("_Prog_Lav2_Temperatura")
   			Case 17
   				SmartTags("Lav4_Prog"&progStr&"_EnjFin_Cant") = SmartTags("_Prog_EnjFin_Cant")
   			Case 18
   				SmartTags("Lav4_Prog"&progStr&"_EnjFin_Tiempo") = SmartTags("_Prog_EnjFin_Tiempo")
   			Case 19
   				SmartTags("Lav4_Prog"&progStr&"_Centr_Tiempo") = SmartTags("_Prog_Centr_Tiempo")
   							
   		End Select 
   		
   		
   End Select
   
   If Err.Number <> 0 Then
   	bfde4b54-0db7-4817-8032-87127bf19bb9 "S600_Problemas para escribir los datos. Error #" & Err.Number & ":'" & Err.Description & "'"
   	Err.Clear
   	Exit Sub
   End If

VB script "SA5_email_SnsPlancha"
   If SmartTags("Alarmas_PL1-Fall-SnsDer") = True Or SmartTags("Alarmas_PL1-Fall-SnsIzq")= True Or SmartTags("Alarmas_PL1-Fall-SnsMed") = True Or SmartTags("Alarmas_PL2-Fall-SnsDer")= True Or SmartTags("Alarmas_PL2-Fall-SnsIzq") = True Or SmartTags("Alarmas_PL2-Fall-SnsMed") Then
   	Dim appOutlook 'As OUTLOOK.APPLICATION
   	Dim mlNewMail 'As MailItem
   	Dim objEntry
   	Dim Text
   	
   	Const addressee = "crj@eprocsrl.com.ar; danielst@live.com.ar;"' josemariacullen@hotmail.com; zekeserio@hotmail.com;"	
   	
   	
   			
   		' Text to be sent 
   		
   		Text = "AVISO SENSOR TAPADO DE PLANCHADORA " + CStr(nro) +" SENSOR " + sns + vbCrLf +_
   				"Hora: " + CStr(Date()) + " "
   				
   		
   		Set appOutlook = CreateObject("OUTLOOK.APPLICATION")
   		
   		
   		'Generating and sending an e-mail:
   		Set mlNewMail = appOutlook.CreateItem(0)
   		mlNewMail.Display
   		mlNewMail.To = addressee
   		mlNewMail.Subject = "AVISO SENSOR TAPADO DE PLANCHADORA " + CStr(nro) +" SENSOR " + sns
   		mlNewMail.Body = Text
   		mlNewMail.save
   		mlNewMail.send 
   		
   		
   	End If

VB script "S601_Actualizar_Vars_Todos"
   Dim progStr, lavnro
   
   If Lav = 1 Then
   		progStr = CStr(SmartTags("_Prog_aModifBraun"))
   		
   		If SmartTags("Lav1_Prog"&progStr&"_EnjFin_Cant") <> 0 Then
   			lavnro = "1"
   			
   		ElseIf SmartTags("Lav2_Prog"&progStr&"_EnjFin_Cant") <> 0 Then
   		
   		lavnro = "2"
   		ElseIf SmartTags("Lav3_Prog"&progStr&"_EnjFin_Cant") <> 0 Then
   				
   		lavnro = "3"
   		
   		End If		
   				SmartTags("_Prog_EnjIni_Cant") = SmartTags("Lav"&lavnro&"_Prog"&progStr&"_EnjIni_Cant")
   
   				SmartTags("_Prog_EnjIni_Tiempo") = SmartTags("Lav"&lavnro&"_Prog"&progStr&"_EnjIni_Tiempo")
   
   				SmartTags("_Prog_EnjIni_NivAg") = SmartTags("Lav"&lavnro&"_Prog"&progStr&"_EnjIni_NivAg")
   
   				SmartTags("_Prog_PreLav_Tiempo") = SmartTags("Lav"&lavnro&"_Prog"&progStr&"_PreLav_Tiempo")
   
   				SmartTags("_Prog_PreLav_NivAg") = SmartTags("Lav"&lavnro&"_Prog"&progStr&"_PreLav_NivAg")
   
   				SmartTags("_Prog_PreLav_AgCaliente") = SmartTags("Lav"&lavnro&"_Prog"&progStr&"_PreLav_AgCaliente")
   
   				SmartTags("_Prog_PreLav_Vapor") = SmartTags("Lav"&lavnro&"_Prog"&progStr&"_PreLav_Vapor")
   
   				SmartTags("_Prog_PreLav_Temperatura") = SmartTags("Lav"&lavnro&"_Prog"&progStr&"_PreLav_Temperatura")
   
   				SmartTags("_Prog_Lav1_Tiempo") = SmartTags("Lav"&lavnro&"_Prog"&progStr&"_Lav1_Tiempo")
   
   				SmartTags("_Prog_Lav1_NivAg") = SmartTags("Lav"&lavnro&"_Prog"&progStr&"_Lav1_NivAg")
   
   				SmartTags("_Prog_Lav1_AgCaliente") = SmartTags("Lav"&lavnro&"_Prog"&progStr&"_Lav1_AgCaliente")
   
   				SmartTags("_Prog_Lav1_Temperatura") = SmartTags("Lav"&lavnro&"_Prog"&progStr&"_Lav1_Temperatura")
   
   				SmartTags("_Prog_Lav2_Tiempo") = SmartTags("Lav"&lavnro&"_Prog"&progStr&"_Lav2_Tiempo")
   
   				SmartTags("_Prog_Lav2_NivAg") = SmartTags("Lav"&lavnro&"_Prog"&progStr&"_Lav2_NivAg")
   
   				SmartTags("_Prog_Lav2_AgCaliente") = SmartTags("Lav"&lavnro&"_Prog"&progStr&"_Lav2_AgCaliente")
   
   				SmartTags("_Prog_Lav2_Temperatura") = SmartTags("Lav"&lavnro&"_Prog"&progStr&"_Lav2_Temperatura")
   
   				SmartTags("_Prog_EnjFin_Cant") = SmartTags("Lav"&lavnro&"_Prog"&progStr&"_EnjFin_Cant")
   
   				SmartTags("_Prog_EnjFin_Tiempo") = SmartTags("Lav"&lavnro&"_Prog"&progStr&"_EnjFin_Tiempo")
   
   				SmartTags("_Prog_Centr_Tiempo") = SmartTags("Lav"&lavnro&"_Prog"&progStr&"_Centr_Tiempo")
   
   
   If Err.Number <> 0 Then
   	bfde4b54-0db7-4817-8032-87127bf19bb9 "S601_Problemas para escribir los datos. Error 1#" & Err.Number & ":'" & Err.Description & "'"
   	Err.Clear
   	Exit Sub
   End If
   
   End If
   
   If Lav = 2 Then
   	
   			progStr = CStr(SmartTags("_Prog_aModifGirbau"))
   
   				SmartTags("_Prog_EnjIni_Cant") = SmartTags("Lav4_Prog"&progStr&"_EnjIni_Cant")
   
   				SmartTags("_Prog_EnjIni_Tiempo") = SmartTags("Lav4_Prog"&progStr&"_EnjIni_Tiempo")
   
   				SmartTags("_Prog_EnjIni_NivAg") = SmartTags("Lav4_Prog"&progStr&"_EnjIni_NivAg")
   
   				SmartTags("_Prog_PreLav_Tiempo") = SmartTags("Lav4_Prog"&progStr&"_PreLav_Tiempo")
   
   				SmartTags("_Prog_PreLav_NivAg") = SmartTags("Lav4_Prog"&progStr&"_PreLav_NivAg")
   
   				SmartTags("_Prog_PreLav_AgCaliente") = SmartTags("Lav4_Prog"&progStr&"_PreLav_AgCaliente")
   
   				SmartTags("_Prog_PreLav_Vapor") = SmartTags("Lav4_Prog"&progStr&"_PreLav_Vapor")
   
   				SmartTags("_Prog_PreLav_Temperatura") = SmartTags("Lav4_Prog"&progStr&"_PreLav_Temperatura")
   
   				SmartTags("_Prog_Lav1_Tiempo") = SmartTags("Lav4_Prog"&progStr&"_Lav1_Tiempo")
   
   				SmartTags("_Prog_Lav1_NivAg") = SmartTags("Lav4_Prog"&progStr&"_Lav1_NivAg")
   
   				SmartTags("_Prog_Lav1_AgCaliente") = SmartTags("Lav4_Prog"&progStr&"_Lav1_AgCaliente")
   
   				SmartTags("_Prog_Lav1_Temperatura") = SmartTags("Lav4_Prog"&progStr&"_Lav1_Temperatura")
   
   				SmartTags("_Prog_Lav2_Tiempo") = SmartTags("Lav4_Prog"&progStr&"_Lav2_Tiempo")
   
   				SmartTags("_Prog_Lav2_NivAg") = SmartTags("Lav4_Prog"&progStr&"_Lav2_NivAg")
   
   				SmartTags("_Prog_Lav2_AgCaliente") = SmartTags("Lav4_Prog"&progStr&"_Lav2_AgCaliente")
   
   				SmartTags("_Prog_Lav2_Temperatura") = SmartTags("Lav4_Prog"&progStr&"_Lav2_Temperatura")
   
   				SmartTags("_Prog_EnjFin_Cant") = SmartTags("Lav4_Prog"&progStr&"_EnjFin_Cant")
   
   				SmartTags("_Prog_EnjFin_Tiempo") = SmartTags("Lav4_Prog"&progStr&"_EnjFin_Tiempo")
   
   				SmartTags("_Prog_Centr_Tiempo") = SmartTags("Lav4_Prog"&progStr&"_Centr_Tiempo")
   				
   If Err.Number <> 0 Then
   	bfde4b54-0db7-4817-8032-87127bf19bb9 "S601_Problemas para escribir los datos. Error 2#" & Err.Number & ":'" & Err.Description & "'"
   	Err.Clear
   	Exit Sub
   End If
   	
   End If

scheduled task "Gen_Inf_Lavadoras"
   on Action: "S403_ActDia"(); "S20_Generador_Inf"()

scheduled task "ActualizarDia"
   on Action: "S403_ActDia"()

scheduled task "Gen_Inf_Mensual"
   on Action: "S404_ActMes"(); "S500_InformePeriodico"(1, "Inf_Ano", "Inf_Mes")

scheduled task "Gen_Inf_Anual"
   on Action: "S405_ActAno"(); "S500_InformePeriodico"(2, 0, "Inf_Ano")

scheduled task "Actualizacion Grafica"
   Triggers <- "1 min"
*)

(* ===== HMI "HMI_RT_2" =====
system functions are stored by id; their names below are inferred from use
connection "HMI_Conexión_3": ETHERNET, SMART_S7_1200_OMS

HMI tags "Tabla de variables estándar"
   "Planchadora1_Supervisores[1].Estado" : Bool = PLC Planchadora1.Supervisores[4].Estado, 1 s
   "Planchadora1_Supervisores[2].Estado" : Bool = PLC Planchadora1.Supervisores[2].Estado, 1 s
   "Planchadora1_Supervisores[3].Estado" : Bool = PLC Planchadora1.Supervisores[3].Estado, 1 s
   "Planchadora1_Supervisores[4].Estado" : Bool = PLC Planchadora1.Supervisores[4].Estado, 1 s
   "Planchadora1_Operadores[1].Estado" : Bool = PLC Planchadora1.Operadores[1].Estado, 1 s
   "Planchadora1_Operadores[2].Estado" : Bool = PLC Planchadora1.Operadores[2].Estado, 1 s
   "Planchadora1_Operadores[4].Estado" : Bool = PLC Planchadora1.Operadores[4].Estado AT %DB1.DBX0.0, 1 s
   "Planchadora1_Operadores[3].Estado" : Bool = PLC Planchadora1.Operadores[3].Estado AT %DB1.DBX0.0, 1 s
   "Planchadora1_Operadores[5].Estado" : Bool = PLC Planchadora1.Operadores[5].Estado AT %DB1.DBX0.0, 1 s
   "Planchadora1_Operadores[6].Estado" : Bool = PLC Planchadora1.Operadores[6].Estado AT %DB1.DBX0.0, 1 s
   "Planchadora1_Operadores[7].Estado" : Bool = PLC Planchadora1.Operadores[7].Estado AT %DB1.DBX0.0, 1 s
   "Planchadora1_Operadores[8].Estado" : Bool = PLC Planchadora1.Operadores[8].Estado AT %DB1.DBX0.0, 1 s
   "Planchadora1_Operadores[9].Estado" : Bool = PLC Planchadora1.Operadores[9].Estado AT %DB1.DBX0.0, 1 s
   "Planchadora1_Operadores[10].Estado" : Bool = PLC Planchadora1.Operadores[10].Estado AT %DB1.DBX0.0, 1 s
   "Planchadora1_EstadoSsIzq" : Byte = PLC Planchadora1.EstadoSsIzq, 1 s
   "Planchadora1_EstadoSSMed" : Byte = PLC Planchadora1.EstadoSSMed, 1 s
   "Planchadora1_EstadoSsDer" : Byte = PLC Planchadora1.EstadoSsDer, 1 s
   "Planchadora1_SumaOperario" : Int = PLC Planchadora1.SumaOperario, 1 s

Template "Plantilla_1" 320x240
   GraphicView "Plantilla_Visor de gráficos_1" at 85,0 size 20x20; Picture "123"
   GraphicView "Plantilla_Visor de gráficos_2" at 105,3 size 96x16; Picture "456"
   TextField "Plantilla_Campo de texto_1" at 224,2 size 87x16; Text 'Planchadoras'
   GraphicView "Plantilla_Visor de gráficos_3" at 47,0 size 36x20; Picture "213"
   GraphicView "Plantilla_Visor de gráficos_4" at 0,2 size 48x17; Picture "1231"

screen "Principal" 320x240, template "Plantilla_1"
   Button "Salir" at 241,200 size 52x40; TextOn 'Salir'; TextOff 'Salir'; PictureOn "ExitRuntime_KTP400_Basic_mono_PN"; PictureOff "ExitRuntime_KTP400_Basic_mono_PN"; Authorization "Operación"
      on Release: StopRuntime(0)
   IOField "Campo ES_1" at 86,104 size 136x79; FormatPattern 99
      ProcessValue <- "Planchadora1_SumaOperario"
   TextField "Campo de texto_1" at 52,52 size 75x32; Text 'Turno'
   TextField "Campo de texto_2" at 148,52 size 101x32; Text 'Mañana'
      Visibility <- "Planchadora1_Supervisores[1].Estado"
   TextField "Campo de texto_3" at 148,52 size 74x32; Text 'Tarde'
      Visibility <- "Planchadora1_Supervisores[2].Estado"
   TextField "Campo de texto_4" at 148,52 size 80x32; Text 'Noche'
      Visibility <- "Planchadora1_Supervisores[3].Estado"
   TextField "Campo de texto_5" at 148,52 size 57x32; Text 'Otro'
      Visibility <- "Planchadora1_Supervisores[4].Estado"
*)

(* ===== HMI "HMI_RT_1" =====

ScreenModuleEditorView "CheckBox_Valido" 640x480
   TextField "Campo de texto_41" at 10,10 size 32x32; Text 'X'
   Group "Group_20" at 10,10 size 32x32
   Button "Botón_13" at 10,10 size 32x32; TextOff 'Text'
*)

(* ===== HMI "HMI_RT_1" =====
system functions are stored by id; their names below are inferred from use

HMI tags "Tabla de variables estándar"
   "Cambiar" : Bool, internal
   "Valido" : Bool, internal

ScreenModuleEditorView "CheckBox_Valido" 640x480
   TextField "Campo de texto_41" at 10,10 size 32x32; Text 'X'
   Group "Group_20" at 10,10 size 32x32
   Button "Botón_13" at 10,10 size 32x32; TextOff 'Text'
      on Click: InvertBit("Estado")
   Rectangle "Rectángulo_23" at 10,10 size 32x32
      Visibility <- "Estado"
*)

(* ===== HMI "HMI_RT_1" =====
system functions are stored by id; their names below are inferred from use

ScreenModuleEditorView "CheckBox_Valido" 640x480
   TextField "Campo de texto_41" at 10,10 size 32x32; Text 'X'
   Group "Group_20" at 10,10 size 32x32
   Button "Botón_13" at 10,10 size 32x32; TextOff 'Text'
      on Click: InvertBit(N)
   Rectangle "Rectángulo_23" at 10,10 size 32x32
      Visibility <- "Estado"
*)

(* ===== HMI "HMI_RT_1" =====

HMI tags "Tabla de variables estándar"
   "Estado" : Bool, internal

ScreenModuleEditorView "CheckBox_Valido" 640x480
   TextField "Campo de texto_41" at 10,10 size 32x32; Text 'X'
   Group "Group_20" at 10,10 size 32x32
   Button "Botón_13" at 10,10 size 32x32; TextOff 'Text'
   Rectangle "Rectángulo_23" at 10,10 size 32x32
      Visibility <- "Estado"
   Polygon "Polígono_23" at 14,13 size 23x24
      Visibility <- "Estado"
*)

(* ===== HMI "HMI_RT_1" =====

HMI tags "Tabla de variables estándar"
   "Estado" : Bool, internal

ScreenModuleEditorView "CheckBox_Valido" 640x480
   TextField "Campo de texto_41" at 10,10 size 32x32; Text 'X'
   Group "Group_20" at 10,10 size 32x32
   Button "Botón_13" at 10,10 size 32x32; TextOff 'Text'
   Rectangle "Rectángulo_23" at 10,10 size 32x32
      Visibility <- "Estado"
   Polygon "Polígono_23" at 14,13 size 23x24
      Visibility <- "Estado"
*)

(* ===== HMI "HMI_RT_1" =====

HMI tags "Tabla de variables estándar"
   "Estado" : Bool, internal

ScreenModuleEditorView "CheckBox_Valido" 640x480
   TextField "Campo de texto_41" at 10,10 size 32x32; Text 'X'
   Group "Group_20" at 10,10 size 32x32
   Button "Botón_13" at 10,10 size 32x32; TextOff 'Text'
   Rectangle "Rectángulo_23" at 10,10 size 32x32
      Visibility <- "EstadoValido"
   Polygon "Polígono_23" at 14,13 size 23x24
      Visibility <- "EstadoValido"
*)

(* ===== HMI "HMI_RT_1" =====

HMI tags "Tabla de variables estándar"
   "Estado" : Bool, internal

ScreenModuleEditorView "CheckBox_Valido" 640x480
   TextField "Campo de texto_41" at 10,10 size 32x32; Text 'X'
   Group "Group_20" at 10,10 size 32x32
   Button "Botón_13" at 10,10 size 32x32; TextOff 'Text'
   Rectangle "Rectángulo_23" at 10,10 size 32x32
      Visibility <- "EstadoValido"
   Polygon "Polígono_23" at 14,13 size 23x24
      Visibility <- "EstadoValido"
*)

(* ===== HMI "HMI_RT_1" =====

HMI tags "Tabla de variables estándar"
   "Estado" : Bool, internal

ScreenModuleEditorView "CheckBox_Valido" 640x480
   TextField "Campo de texto_41" at 10,10 size 32x32; Text 'X'
   Group "Group_20" at 10,10 size 32x32
   Button "Botón_13" at 10,10 size 32x32; TextOff 'Text'
   Rectangle "Rectángulo_23" at 10,10 size 32x32
      Visibility <- "EstadoValido"
   Polygon "Polígono_23" at 14,13 size 23x24
      Visibility <- "EstadoValido"
*)